// Interface implemented by device FBs and consumed by FB_SparkplugSession
// to orchestrate the birth cycle and device lifecycle.
INTERFACE I_SparkplugDevice

// Called by the session at the start of each birth cycle, after NBIRTH is sent.
// The device must encode and publish its DBIRTH using the session's
// GetNextSeq() and Publish() methods.
METHOD OnBirth
END_METHOD

// Encodes and publishes a DDATA message using the current metric values.
// Returns FALSE if the session is not online or the publish fails.
METHOD PublishData : BOOL
VAR_INPUT
	bChangedOnly		: BOOL  := FALSE;
END_VAR
END_METHOD

// Publishes a DDEATH for this device, signalling the host that it is offline.
// Returns FALSE if the session is not online or the publish fails.
METHOD PublishDeath : BOOL
END_METHOD

// Called by the session when the device is registered via AddDevice.
// The device stores the session reference and device ID for use in OnBirth/PublishData.
METHOD SetSession
VAR_INPUT
	sDeviceId	: STRING(127);
	ipSession	: I_SparkplugSession;
END_VAR
END_METHOD

END_INTERFACE

(* stored: Version 1.1.0.1
   Itf I_SparkplugDevice: Id {33333333-0000-0000-0000-000000000001}
   Method OnBirth: Id {33333333-0000-0000-0000-000000000011}
   Method PublishData: Id {33333333-0000-0000-0000-000000000012}
   Method PublishDeath: Id {33333333-0000-0000-0000-000000000013}
   Method SetSession: Id {33333333-0000-0000-0000-000000000010} *)
